INTERFACE IIntersectionController EXTENDS TOF_Automation.IAutomationController

{attribute 'monitoring' := 'call'}
PROPERTY FINAL AdjustSpeedButton : TOF_Devices_IO.IDigitalInput
GET
END_GET
END_PROPERTY

{attribute 'monitoring' := 'call'}
PROPERTY FINAL LightsState : INTERSECTION_LIGHTS_STATE
GET
END_GET
END_PROPERTY

{attribute 'monitoring' := 'call'}
PROPERTY FINAL Mode : INTERSECTION_MODE
GET
END_GET
END_PROPERTY

{attribute 'monitoring' := 'call'}
PROPERTY FINAL ResetButton : TOF_Devices_IO.IDigitalInput
GET
END_GET
END_PROPERTY

METHOD SetSwitchingSpeedCorrectionPercent
VAR_INPUT
	correctionPercent : SPEED_CORRECTION_PERCENT;
END_VAR
END_METHOD

METHOD SetYellowFlashingModeOff
END_METHOD

{attribute 'monitoring' := 'call'}
PROPERTY FINAL SetYellowFlashingModeOffButton : TOF_Devices_IO.IDigitalInput
GET
END_GET
END_PROPERTY

METHOD SetYellowFlashingModeOn
END_METHOD

{attribute 'monitoring' := 'call'}
PROPERTY FINAL SetYellowFlashingModeOnButton : TOF_Devices_IO.IDigitalInput
GET
END_GET
END_PROPERTY

{attribute 'monitoring' := 'call'}
PROPERTY FINAL SignalGroup1 : REFERENCE TO
	ARRAY [1..IntersectionConstants.TRAFFIC_LIGHTS_PER_GROUP] OF IReadOnlyTrafficLight
GET
END_GET
END_PROPERTY

{attribute 'monitoring' := 'call'}
PROPERTY FINAL SignalGroup2 : REFERENCE TO
	ARRAY [1..IntersectionConstants.TRAFFIC_LIGHTS_PER_GROUP] OF IReadOnlyTrafficLight
GET
END_GET
END_PROPERTY

{attribute 'monitoring' := 'call'}
PROPERTY FINAL SwitchingSpeedCorrectionPercent : SPEED_CORRECTION_PERCENT
GET
END_GET
END_PROPERTY

{attribute 'monitoring' := 'call'}
PROPERTY FINAL SwitchSpeedAdjuster : TOF_Devices_IO.IAnalogInput
GET
END_GET
END_PROPERTY

METHOD ThrowExceptionInDemoExceptionGenerator
VAR_IN_OUT CONSTANT
	exceptionMessage : STRING(255);
	isCritical : BOOL; 
END_VAR
END_METHOD

{attribute 'monitoring' := 'call'}
PROPERTY FINAL TrafficLights : REFERENCE TO ARRAY [1..IntersectionConstants.TOTAL_TRAFFIC_LIGHTS] OF IReadOnlyTrafficLight
GET
END_GET
END_PROPERTY

METHOD TurnOff
END_METHOD

{attribute 'monitoring' := 'call'}
PROPERTY FINAL TurnOffButton : TOF_Devices_IO.IDigitalInput
GET
END_GET
END_PROPERTY

METHOD TurnOn
END_METHOD

{attribute 'monitoring' := 'call'}
PROPERTY FINAL TurnOnButton : TOF_Devices_IO.IDigitalInput
GET
END_GET
END_PROPERTY

END_INTERFACE

(* stored: Version 1.1.0.1
   Itf IIntersectionController: Id {28647d84-1ce3-4815-a390-9e82e485caf1}
   Folder Commands: Id {9fe5f94b-6d49-4e08-8469-d5af3d174eb3}
   Folder Statuses: Id {e19a8bf6-6de5-43b9-99e8-aa87b4b3ac22}
   Folder Subdevices: Id {52172a49-dc23-4784-8a34-642732a4f005}
   Property AdjustSpeedButton: Id {09a701f3-c822-4b73-9409-1a50bb968c71}
   Get Get: Id {f79d1a29-830e-41e8-9ab9-2288ea847682}
   Property LightsState: Id {86b37f47-f060-4fbf-8eb9-3fce5da737fc}
   Get Get: Id {5c2203e5-3314-4b79-b87c-5831f684c812}
   Property Mode: Id {8770cd46-3029-49d7-8b6d-f81bba200339}
   Get Get: Id {dade3d60-724e-455d-842b-cb8ad4926992}
   Property ResetButton: Id {0ab6b873-398b-4883-99a2-5e028d5b5cdc}
   Get Get: Id {8de62190-aa46-4133-9f70-4a458b75dcf2}
   Method SetSwitchingSpeedCorrectionPercent: Id {dd8def6d-b3a3-4b73-98b2-8a590327f7b0}
   Method SetYellowFlashingModeOff: Id {4c2122f0-0e96-48b0-9aa3-6c9b8aff6ab9}
   Property SetYellowFlashingModeOffButton: Id {653fa861-0898-4d9b-82b7-29e601d185a2}
   Get Get: Id {71811033-68e4-4bc9-8ef4-f591356f63f3}
   Method SetYellowFlashingModeOn: Id {41154cb2-21a1-48c7-8faa-2b7368fcd741}
   Property SetYellowFlashingModeOnButton: Id {f66d0dd9-83b9-4109-aeff-116f2a705f1a}
   Get Get: Id {7beeed40-ef9b-4eb8-b14e-c0385ddcac59}
   Property SignalGroup1: Id {7ae7073d-f3ff-473f-952d-419685b15664}
   Get Get: Id {f0e55ebf-7c74-4674-b281-7bf20ca3c076}
   Property SignalGroup2: Id {45c4f515-dc70-4e95-9beb-aeece2b386dd}
   Get Get: Id {582f6a6c-e339-4263-976b-9da7cb94f4af}
   Property SwitchingSpeedCorrectionPercent: Id {fcd875cd-6a57-41a0-bf6d-8004bf2f90de}
   Get Get: Id {a8a6111b-17a9-40bf-98d0-2672915bf414}
   Property SwitchSpeedAdjuster: Id {e9fca1a2-9c43-40f7-be78-4e15cdfbdb1b}
   Get Get: Id {ca0ceb73-1d23-4f80-8f0e-911b055b83a3}
   Method ThrowExceptionInDemoExceptionGenerator: Id {9e6aea40-70f1-469b-8846-298be146f806}
   Property TrafficLights: Id {7b1f3c2b-dfc7-4373-85aa-9174e04f9904}
   Get Get: Id {710bf72e-b285-4274-88cc-f0e90d94a3c6}
   Method TurnOff: Id {0c089be5-a16b-434c-82c5-646302b8c882}
   Property TurnOffButton: Id {3c472fd2-12d0-47de-a515-0fbc83482029}
   Get Get: Id {1133c40f-7199-4f29-a073-6df267eba772}
   Method TurnOn: Id {d6179d65-edb5-4d14-8839-d9b0547d39a2}
   Property TurnOnButton: Id {2cc5f4ed-614f-41e5-93d1-020adf400cb2}
   Get Get: Id {538fd1e0-6988-4bca-88e0-dec2e282afc3} *)
